PROGRAM B_Program
VAR
	i : UINT;
	x : LREAL;
	x_inc : LREAL := 0.0001;
	cyclecount : UINT;
END_VAR

cyclecount := cyclecount + 1;

IF cyclecount > 10 THEN
	FOR i := 0 TO 1000 DO
		x := x + x_inc;
	END_FOR	
	cyclecount := 0;
END_IF

END_PROGRAM

(* stored: Version 1.1.0.1, ProductVersion 3.1.4025.12
   POU B_Program: Id {e7957ae7-cb23-4536-a265-606f38247fcb}, SpecialFunc None *)
